// TIA Portal V20 export
DATA_BLOCK "DB_LightsManagement"   // DB500
// stored: AutoNumber false, InstanceOfName FB_LightsManagement, InstanceOfType FB
"FB_LightsManagement"
BEGIN
END_DATA_BLOCK
